(* CoDeSys 2.3.9.41 project: 123.pro *)
(* Libraries: STANDARD.LIB 4.10.05 11:14:46, IECSFC.LIB 13.4.06 15:51:28, SYSLIBTIME.LIB 20.2.06 13:31:16, SYSTASKINFO.LIB 20.2.06 13:31:38, ANALYZATION.LIB 5.10.99 09:05:06, SYSLIBCALLBACK.LIB 20.2.06 13:31:08 *)

(* PLC configuration (modules and I/O channels)
Fast discrete inputs [I_SIMPLE_INPUT] node 0, in %IB0 out %QB0 {Filtrationtime = 10; Visibility = No}
  AT %IX0.0 [BitInput] Discrete input 1
  AT %IX0.1 [BitInput] Discrete input 2
x AT %IB1.0 [ByteInput] 8 discrete inputs
z AT %IB1.1 [ByteInput] 8 discrete inputs
Fast discrete outputs [OWEN_ID570] node 2, in %IB2 out %QB2 {SafeValueBool = FALSE; SafeValueBool = FALSE; SafeValueBool = FALSE; SafeValueBool = FALSE; Visibility = No}
  AT %QX2.0 [BitOutput] Fast discrete output 1
  AT %QX2.1 [BitOutput] Fast discrete output 2
  AT %QX2.2 [BitOutput] Fast discrete output 3
  AT %QX2.3 [BitOutput] Fast discrete output 4
y AT %QB3.0 [ByteOutput] 8 discrete outputs
q AT %QB3.1 [ByteOutput] 2 discrete outputs
Special input [ID103] node 4, in %IB4 out %QB4 {Filtrationtime = 1000; PinCount = 1; WatchDogPeriod = 400; PollPeriod = 3000; Visibility = No}
  AT %IX4.0 [BitInput] Special input
Special output [ID104] node 5, in %IB5 out %QB5 {Visibility = No; PinCount = 1}
  AT %QX5.0 [BitOutput] Special output
TCP [TCP_ID221] node 0, in %IB6.0.0 out %QB6.0.0 {RemotePort = 502; Visibility = No}
v AT %QB6.1.0 [ByteOutput]
w AT %QB6.2.0 [ByteOutput]
c AT %QW6.3.0 [WordOutput]
d AT %QW6.4.0 [WordOutput]
*)

(* POU PLC_PRG, LD *)
PROGRAM PLC_PRG
VAR
	www: TON;
	n: TIME;
	sofiko: TON;
	m: BOOL;
	rr: TIME;
	matviko: TOF;
	lll: TIME;
	tikitikitiki: TIME;
	pppp: TIME;
END_VAR
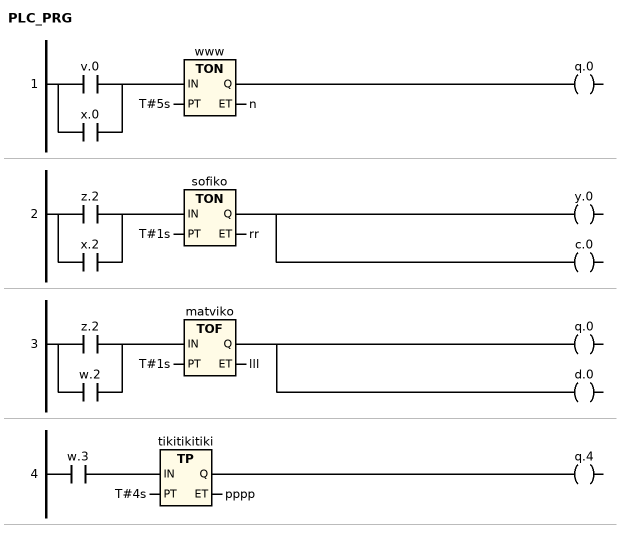
_LD_ (* Ladder Diagram *)
NETWORK 1
	{ [v.0] | [x.0] } - www:TON(IN: *, PT: T#5s, ET => n) --- (q.0)
NETWORK 2
	{ [z.2] | [x.2] } - sofiko:TON(IN: *, PT: T#1s, ET => rr) --- (y.0) (c.0)
NETWORK 3
	{ [z.2] | [w.2] } - matviko:TOF(IN: *, PT: T#1s, ET => lll) --- (q.0) (d.0)
NETWORK 4
	[w.3] - tikitikitiki:TP(IN: *, PT: T#4s, ET => pppp) --- (q.4)
_END_LD_
(* the same logic as Structured Text *)
(* Network 1 *)
www(IN := v.0 OR x.0, PT := T#5s);
n := www.ET;
q.0 := www.Q;
(* Network 2 *)
sofiko(IN := z.2 OR x.2, PT := T#1s);
rr := sofiko.ET;
y.0 := sofiko.Q;
c.0 := sofiko.Q;
(* Network 3 *)
matviko(IN := z.2 OR w.2, PT := T#1s);
lll := matviko.ET;
q.0 := matviko.Q;
d.0 := matviko.Q;
(* Network 4 *)
tikitikitiki(IN := w.3, PT := T#4s);
pppp := tikitikitiki.ET;
q.4 := tikitikitiki.Q;
END_PROGRAM
